(* Logix 5000 project; controller EuniceF_ICA16 vendor 1 type 14 code 150 rev 37.11; software revision 37.00 *)

TASK MainTask (continuous, watchdog 500 ms) : MainProgram

MODULES
   Local : vendor 1 type 14 code 150 (Compact 0, rev 37.11)
      Discrete_IO : Embedded (Compact 1, rev 3.1, Output RPI 20 ms)
      Analog_IO : Embedded (Compact 2, rev 1.1, Output RPI 80 ms)
      Counters : Embedded (Compact 3, rev 1.1, Output RPI 20 ms)
END_MODULES

VAR_GLOBAL   (* controller tags *)
   Motor : ALIAS FOR Local:1:O.Data.1;
   Reset : ALIAS FOR Local:1:I.Data.0;
   seq : DINT;
   START : ALIAS FOR Local:1:I.Data.14;
   StartCount : COUNTER;
   STEP : ALIAS FOR Local:1:I.Data.12;
   StepCount : COUNTER;
   STOP : ALIAS FOR Local:1:I.Data.9;
END_VAR

PROGRAM MainProgram   (* main routine MainRoutine *)

ROUTINE MainRoutine   (* ladder *)
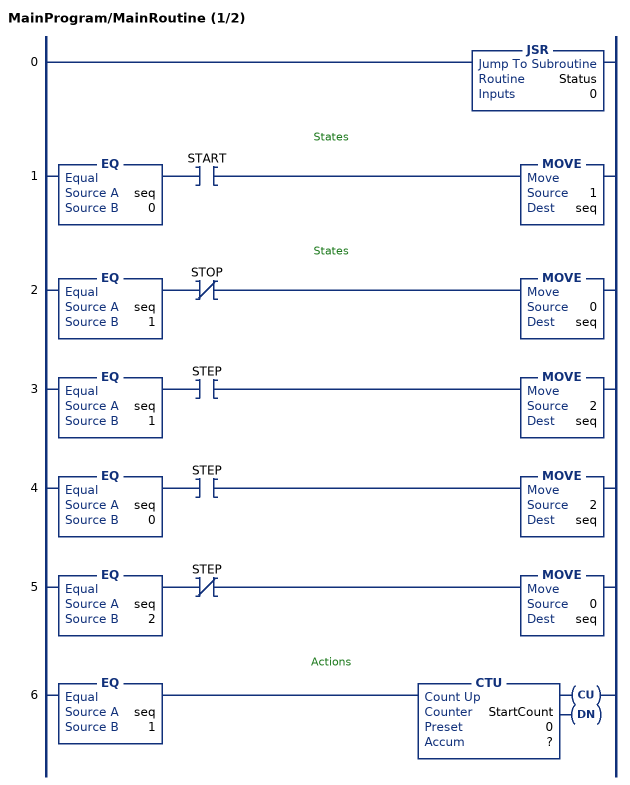
   0: JSR(Status,0);
   // States
   1 (stored rung type 13): EQ(seq,0)XIC(START)MOVE(1,seq);
   // States
   2: EQ(seq,1)XIO(STOP)MOVE(0,seq);
   3: EQ(seq,1)XIC(STEP)MOVE(2,seq);
   4: EQ(seq,0)XIC(STEP)MOVE(2,seq);
   5: EQ(seq,2)XIO(STEP)MOVE(0,seq);
   // Actions
   6: EQ(seq,1)CTU(StartCount,?,?);
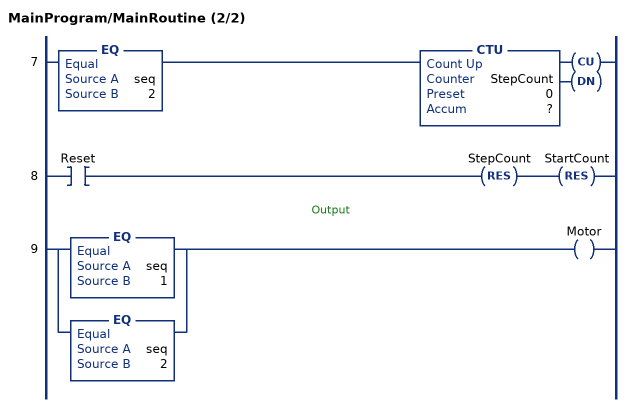
   7: EQ(seq,2)CTU(StepCount,?,?);
   8: XIC(Reset)RES(StepCount)RES(StartCount);
   // Output
   9: [EQ(seq,1) ,EQ(seq,2) ]OTE(Motor);
END_ROUTINE

ROUTINE Status   (* structured text *)
   
END_ROUTINE
END_PROGRAM
